KUKA KRL data list: Functions.dat

&ACCESS RV
&REL 2
DEFDAT Functions PUBLIC

ENDDAT
